// TwinCAT 3 PLC project PLC
// ProgramVersion: 3.1.4026.22
// libraries:
//   Tc2_EtherCAT, * (Beckhoff Automation GmbH)
//   Tc2_Standard, * (Beckhoff Automation GmbH)
//   Tc2_System, * (Beckhoff Automation GmbH)
// project tree:
//   / PlcTask.TcTTO, PlcTask2.TcTTO, PlcTask3.TcTTO
//   POUs/ F_ConsumeTime.TcPOU (not stored), PRG_Task3.TcPOU, PRG_Task1.TcPOU, PRG_Task2.TcPOU
// real-time tasks:
//   TASK PlcTask1: cycle T#10ms, priority 1, ADS port 350
//   TASK PlcTask2: cycle T#10ms, priority 2, ADS port 351
//   TASK PlcTask3: cycle T#10ms, priority 3, ADS port 352

CONFIGURATION PLC
    RESOURCE PLC ON TwinCAT3
        TASK PlcTask(INTERVAL := T#10ms, PRIORITY := 1);
        TASK PlcTask2(INTERVAL := T#10ms, PRIORITY := 2);
        TASK PlcTask3(INTERVAL := T#10ms, PRIORITY := 3);
        PROGRAM PRG_Task1 WITH PlcTask : PRG_Task1;
        PROGRAM PRG_Task2 WITH PlcTask2 : PRG_Task2;
        PROGRAM PRG_Task3 WITH PlcTask3 : PRG_Task3;
    END_RESOURCE
END_CONFIGURATION

// ---- POUs/PRG_Task1.TcPOU
PROGRAM PRG_Task1
VAR
END_VAR

F_ConsumeTime(1000);

END_PROGRAM

// ---- POUs/PRG_Task2.TcPOU
PROGRAM PRG_Task2
VAR
END_VAR

F_ConsumeTime(2000);

END_PROGRAM

// ---- POUs/PRG_Task3.TcPOU
PROGRAM PRG_Task3
VAR
END_VAR

F_ConsumeTime(4000);

END_PROGRAM
